(* IEC 61131-3 sources: plcassist-cli/packages/volt-lsp-iec/test-corpus/bakon-nano/Device/Plc Logic/Application/POUs/LenzeFunctions/XYA_Functions, 3 files *)

(* ---- CalcCheckSWLimit_XYA.fun ---- *)
(***********************************************************************************
Creation: LENL 		Datum: march 2008		Version: 1.0.0
 ***********************************************************************************
 FUNCTION:

check SW limits for XYA

 ***********************************************************************************
Name							Datum				Changes
Kling 							24.03.2009		Implementation

************************************************************************************
NOTE:

***********************************************************************************)

FUNCTION CalcCheckSWLimit_XYA : BOOL
VAR_INPUT
	Point :XYA_Target;
	AxisX :REFERENCE TO AXIS_REF;
	AxisY :REFERENCE TO AXIS_REF;
	AxisA :REFERENCE TO AXIS_REF;
END_VAR
VAR
END_VAR

	CalcCheckSWLimit_XYA:=FALSE;
IF (Point.X_Target < AxisX.lrSWLimitNeg) OR  (Point.X_Target >  AxisX.lrSWLimitPos) OR (Point.Y_Target < AxisY.lrSWLimitNeg) OR 	(Point.Y_Target >  AxisY.lrSWLimitPos) OR (Point.A_Target < AxisA.lrSWLimitNeg) OR  (Point.A_Target >  AxisA.lrSWLimitPos)  THEN
	CalcCheckSWLimit_XYA:=TRUE;
END_IF

END_FUNCTION

(* ---- CalcGearingRatio.fb ---- *)
(***********************************************************************************
Creation: LENL			 		Datum: March 2009			Version: 1.0.0
 ***********************************************************************************
 FUNCTION:

Calculating the gear ratio

 ***********************************************************************************
Name							Datum				Changes					Version
Kling 							24.03.2009		Implementation

************************************************************************************
NOTE:

***********************************************************************************)

FUNCTION_BLOCK CalcGearingRatio
VAR_INPUT
	rMoveMaster:REAL;
	rMoveSlave:REAL;
END_VAR
VAR_OUTPUT
	nGearNum:INT;
	nGearDenum:INT;
	rGearingFactor: REAL;
END_VAR
VAR
	rGearNum: REAL;
	rGearDenum: REAL;
	rGearingFactorABS: REAL;
	bySelect: BYTE;
	rGearNumDir: REAL;
END_VAR

(*Calc gearing-factor*)
IF (rMoveMaster <> 0)  THEN
	rGearingFactor:=rMoveSlave / rMoveMaster;
ELSE
	rGearingFactor:=0;
END_IF

rGearingFactorABS:=ABS(rGearingFactor);

IF rGearingFactorABS <> 0 THEN
	IF rGearingFactorABS > 1 THEN
		rGearNum:=16384;
		rGearDenum:=rGearNum / rGearingFactorABS;
		bySelect:=1;
	ELSE
		rGearDenum:=16384;
		rGearNum:=rGearDenum * rGearingFactorABS;
		bySelect:=2;
	END_IF
ELSE
	rGearNum:=0;
	rGearDenum:=16384;
	bySelect:=3;
END_IF

(*Direction selection*)
IF rGearingFactor < 0 THEN
	rGearNumDir:=-rGearNum;
ELSE
	rGearNumDir:=rGearNum;
END_IF

(*Write to output*)
nGearNum		:=REAL_TO_INT(rGearNumDir);
nGearDenum		:=REAL_TO_INT(rGearDenum);

END_FUNCTION_BLOCK

(* ---- CalcMasterSpeedAcc.fb ---- *)
(***********************************************************************************
Creation: LENL			 		Datum: March 2009			Version: 1.0.0
 ***********************************************************************************
 FUNCTION:

calc max speed of an axis, depending on a variable gear ratio

 ***********************************************************************************
Name							Datum				Changes					Version
Kling 							24.03.2009		Implementation

************************************************************************************
NOTE:

***********************************************************************************)

FUNCTION_BLOCK CalcMasterSpeedAcc
VAR_INPUT
	rGearingRatio:REAL;
END_VAR
VAR_OUTPUT
	rVelocity:REAL;
	rAcceleration:REAL;
END_VAR
VAR
END_VAR

VAR_IN_OUT
	Axis:AXIS_REF;
END_VAR

IF rGearingRatio <> 0 THEN
	rVelocity:=Axis.scPar.MaxVelocity / ABS(rGearingRatio);
	rAcceleration:=Axis.scPar.MaxAcceleration   / ABS(rGearingRatio);
ELSE
	rVelocity:=100000;
	rAcceleration:=10000000;
END_IF

END_FUNCTION_BLOCK
